// TwinCAT 3 PLC project EXAMPLES
// ProgramVersion: 3.1.4024.0
// libraries:
//   Tc2_Standard, * (Beckhoff Automation GmbH)
//   Tc2_System, * (Beckhoff Automation GmbH)
//   Tc3_IotBase, * (Beckhoff Automation GmbH)
//   Tc3_JsonXml, * (Beckhoff Automation GmbH)
//   Tc3_Module, * (Beckhoff Automation GmbH)
// project tree:
//   / PlcTask.TcTTO
//   POUs/ MAIN.TcPOU

CONFIGURATION EXAMPLES
    RESOURCE PLC ON TwinCAT3
        TASK PlcTask(INTERVAL := T#10ms, PRIORITY := 20);
        PROGRAM MAIN WITH PlcTask : MAIN;
    END_RESOURCE
END_CONFIGURATION

// ---- POUs/MAIN.TcPOU
PROGRAM MAIN
VAR
	// Configure JSON and HTTP function blocks 
	fbJson					: FB_JsonDomParser;
	fbHttpClient 			: FB_IotHttpClient:=(
								sHostName:='192.168.0.10',			// Replace with your SPLAY's IP address
								nHostPort:=80,
								bKeepAlive:=TRUE,
								tConnectionTimeout:=T#10S,
								stTLS:=(
									bNoServerCertCheck:=FALSE
								)
							);
							
	// Configure SPLAY function block
	SPLAY					: FB_SPLAY:=(
								fbJson:=fbJson,
								fbHttpClient:=fbHttpClient
							);

	// Main program variables
	nState					: INT:=1;
	jsonReceived			: sJsonValue;
	sReceived				: STRING(10000);		// Output buffer can be any length. Please be aware that some requests in particular will
													// require a larger return/output buffer compared to others, adjust accordingly.
END_VAR

(* 
 * ENTTEC_SPLAY_API LIBRARY EXAMPLES
 *
 *  Commands follow the same naming convention found on the Official SPLAY API.
 *  For additional support, see https://github.com/ENTTEC/SplayApi
 *
 *  The following examples briefly describe the function block usage:
 * 	1: 	Get device information
 *  2: 	Create/update playlist
 *  3: 	Create/save cue
 * 	4: 	Play playlist
 *  5: 	Get cue
*)

CASE nState OF
	
	1:
		// Example 'GET_INFO' command usage
		
		SPLAY.GET_INFO();										// Example of command with no additional parameters
		fbJson.CopyDocument(sReceived, SIZEOF(sReceived));		// Convert JSON object to string output buffer
		ADSLOGSTR(												// Print JSON string to console log
			msgCtrlMask:=ADSLOG_MSGTYPE_STRING,					//  (note: console has a 350 character buffer,
			msgFmtStr:='%s',									//         and will not print for longer messages)
			strArg:=sReceived							
		);
		
		nState:=2;
		
	2:
		// Example 'UPDATE_PLAYLIST' command usage
		
		SPLAY.UPDATE_PLAYLIST(sPlaylist:='{"duration":312000,"timeline":{"track1":{"intensity":100,"cues":[{"start":300000,"name":"Bar Lighting Loop","cue_id":1,"duration":12000,"type":0,"fade":{"in":2000,"out":1500}}]}},"order":1,"intensity":100,"loop":0,"priority":100,"group":0,"start_trigger":{"trigger_id":-1},"stop_trigger":{"trigger_id":-1},"fade_in":3000,"fade_out":2000,"name":"Bar Playlist 1"}');
		fbJson.CopyDocument(sReceived, SIZEOF(sReceived));
		ADSLOGSTR(											
			msgCtrlMask:=ADSLOG_MSGTYPE_STRING,					
			msgFmtStr:='%s',
			strArg:=sReceived				
		);

		nState:=3;
		
	3: 
		// Example 'SAVE_CUE' command usage
		
		SPLAY.SAVE_CUE(sCue:='{"config":{"ch_start":0,"ch_stop":511,"source":1,"universes":[0,1,2,3,4,5,6,7,8,9,10,11,12,13,14,15,16,17,18,19,-1,-1,-1,-1,-1,-1,-1,-1,-1,-1,-1,-1],"trigger":{"type":0}},"cue_id":1,"duration":0,"frames":[[0,0,0,0,0,0,0,0,0,0,0,0,0,0,0,0,0,0,0,0,0,0,0,0,0,0,0,0,0,0,0,0,0,0,0,0,0,0,0,0,0,0,0,0,0,0,0,0,0,0,0,0,0,0,0,0,0,0,0,0,0,0,0,0,0,0,0,0,0,0,0,0,0,0,0,0,0,0,0,0,0,0,0,0,0,0,0,0,0,0,0,0,0,0,0,0,0,0,0,0,0,0,0,0,0,0,0,0,0,0,0,0,0,0,0,0,0,0,0,0,0,0,0,0,0,0,0,0,0,0,0,0,0,0,0,0,0,0,0,0,0,0,0,0,0,0,0,0,0,0,0,0,0,0,0,0,0,0,0,0,0,0,0,0,0,0,0,0,0,0,0,0,0,0,0,0,0,0,0,0,0,0,0,0,0,0,0,0,0,0,0,0,0,0,0,0,0,0,0,0,0,0,0,0,0,0,0,0,0,0,0,0,0,0,0,0,0,0,0,0,0,0,0,0,0,0,0,0,0,0,0,0,0,0,0,0,0,0,0,0,0,0,0,0,0,0,0,0,0,0,0,0,0,0,0,0,0,0,0,0,0,0,0,0,0,0,0,0,0,0,0,0,0,0,0,0,0,0,0,0,0,0,0,0,0,0,0,0,255,255,255,255,255,255,255,255,255,255,255,255,255,255,255,255,255,255,255,255,255,255,255,255,254,254,254,249,249,249,244,244,244,238,238,238,234,234,234,228,228,228,223,223,223,218,218,218,213,213,213,208,208,208,202,202,202,198,198,198,192,192,192,188,188,188,182,182,182,177,177,177,172,172,172,166,166,166,162,162,162,156,156,156,152,152,152,146,146,146,141,141,141,136,136,136,131,131,131,127,127,127,121,121,121,117,117,117,111,111,111,106,106,106,101,101,101,96,96,96,91,91,91,85,85,85,81,81,81,75,75,75,70,70,70,65,65,65,60,60,60,55,55,55,49,49,49,45,45,45,39,39,39,34,34,34,29,29,29,24,24,24,19,19,19,13,13,13,9,9,9,3,3,3,0,0,0,0,0,0,0,0,0,0,0,0,0,0,0,0,0,0,0,0,0,0,0,0,0,0,0,0,0,0,0,0,0,0,0,0,0,0,0,0,0,0,0,0,0,0,0,0,0,0]],"name":"Bar Lighting Loop","type":0}');
		fbJson.CopyDocument(sReceived, SIZEOF(sReceived));
		ADSLOGSTR(												
			msgCtrlMask:=ADSLOG_MSGTYPE_STRING,					
			msgFmtStr:='%s',
			strArg:=sReceived				
		);
		
		nState:=4;
		
	4: 
		// Example 'PLAY' command usage
		
		SPLAY.PLAY(nPlaylistId:=1);								
		fbJson.CopyDocument(sReceived, SIZEOF(sReceived));
		ADSLOGSTR(												
			msgCtrlMask:=ADSLOG_MSGTYPE_STRING,					
			msgFmtStr:='%s',
			strArg:=sReceived					
		);
		
		nState:=5;
		
	5: 
		// Example 'GET_CUE' command usage
		
		SPLAY.GET_CUE(nCueId:=1);
		fbJson.CopyDocument(sReceived, SIZEOF(sReceived));
		ADSLOGSTR(													// Since the return is longer than 350 characters,
			msgCtrlMask:=ADSLOG_MSGTYPE_STRING,						// there will be no output in the console log. 
			msgFmtStr:='%s',
			strArg:=sReceived				
		);															// Try this instead:
		jsonReceived:=fbJson.FindMember(SPLAY.jsonRX, 'cue');		// Search for and return node labelled 'cue'
		jsonReceived:=fbJson.FindMember(jsonReceived, 'name');		// Search for and return node labelled 'name'
		sReceived:=fbJson.GetString(jsonReceived);					// Get string value of specified node
		ADSLOGSTR(													
			msgCtrlMask:=ADSLOG_MSGTYPE_STRING,						 
			msgFmtStr:='%s',
			strArg:=sReceived			
		);
		
		nState:=6;
		
END_CASE

END_PROGRAM
